{attribute addProperty BoxType "ELM9410-0000-0016"}
{attribute addProperty Id "DiagBIT10.1251ErrorBIT10.1252Input_cycle_Counter_BIT_0BIT10.1253Input_cycle_Counter_BIT_1BIT10.1253TxPDO_StateBIT10.1257"}
{attribute addProperty CRC "84631898"}
{attribute addProperty SizeInBites "8"}
{attribute addProperty SizeInBytes "1"}
TYPE Status_050B615A :
STRUCT
	{attribute addProperty Name "Diag"}
	Diag : BIT;
	{attribute addProperty Name "Error"}
	Error : BIT;
	{attribute addProperty Name "Input_cycle_Counter"}
	Input_cycle_Counter_BIT_0 : BIT;
	{attribute addProperty Name "Input_cycle_Counter"}
	Input_cycle_Counter_BIT_1 : BIT;
	{attribute 'hide'}
	reserve_1_BIT_0 : BIT;
	{attribute 'hide'}
	reserve_1_BIT_1 : BIT;
	{attribute addProperty Name "TxPDO_State"}
	TxPDO_State : BIT;
	{attribute 'hide'}
	reserve_2 : BIT;
END_STRUCT
END_TYPE

(* stored: Version 1.2.0.0, ProductVersion 3.1.4024.9
   DUT Status_050B615A: Id {194b28b0-4117-49ab-9950-4badf688ef19} *)
